// TIA Portal project "通信" (V16)

(* hardware
DEVICE "S7-1200 station_1"  S7-1200 Station
   slot 0: "Rack_0"  S7-1200 Rack  Rack  V1.0
   slot 1: "PLC_1"  CPU 1214C DC/DC/DC  6ES7 214-1AG40-0XB0  V4.4
*)

// ===== PLC "PLC_1"  CPU 1214C DC/DC/DC =====

VAR_GLOBAL   // PLC tag table "默认变量表"
   "System_Byte" AT %MB1 : Byte;
   "FirstScan" AT %M1.0 : Bool;
   "DiagStatusUpdate" AT %M1.1 : Bool;
   "AlwaysTRUE" AT %M1.2 : Bool;
   "AlwaysFALSE" AT %M1.3 : Bool;
   "Clock_Byte" AT %MB0 : Byte;
   "Clock_10Hz" AT %M0.0 : Bool;
   "Clock_5Hz" AT %M0.1 : Bool;
   "Clock_2.5Hz" AT %M0.2 : Bool;
   "Clock_2Hz" AT %M0.3 : Bool;
   "Clock_1.25Hz" AT %M0.4 : Bool;
   "Clock_1Hz" AT %M0.5 : Bool;
   "Clock_0.625Hz" AT %M0.6 : Bool;
   "Clock_0.5Hz" AT %M0.7 : Bool;
   "发完成" AT %M100.0 : Bool;
   "接完成" AT %M101.0 : Bool;
END_VAR

DATA_BLOCK "接受DB"   // DB1
{ S7_Optimized_Access := 'FALSE' }
VERSION : 0.1
   VAR
      其他 : Array[0..1] of Byte;
      接收 : Array[0..20] of Byte;
   END_VAR
BEGIN
END_DATA_BLOCK

DATA_BLOCK "传输DB"   // DB2
{ S7_Optimized_Access := 'FALSE' }
VERSION : 0.1
   VAR
      传送DB : Array[0..20] of Byte;
   END_VAR
BEGIN
END_DATA_BLOCK

DATA_BLOCK "数据块_1"   // DB5
{ S7_Optimized_Access := 'FALSE' }
VERSION : 0.1
   VAR
      "1" : Bool;
   END_VAR
BEGIN
END_DATA_BLOCK

ORGANIZATION_BLOCK "Main"   // OB1, LAD, ProgramCycle
TITLE = "Main Program Sweep (Cycle)"
{ S7_Optimized_Access := 'TRUE' }
VERSION : 0.1
   VAR_INPUT
      Initial_Call : Bool;   // Initial call of this OB
      Remanence : Bool;   // =True, if remanent data are available
   END_VAR
BEGIN

REGION Network 2: 传输
   // 先传输，之后接受，在
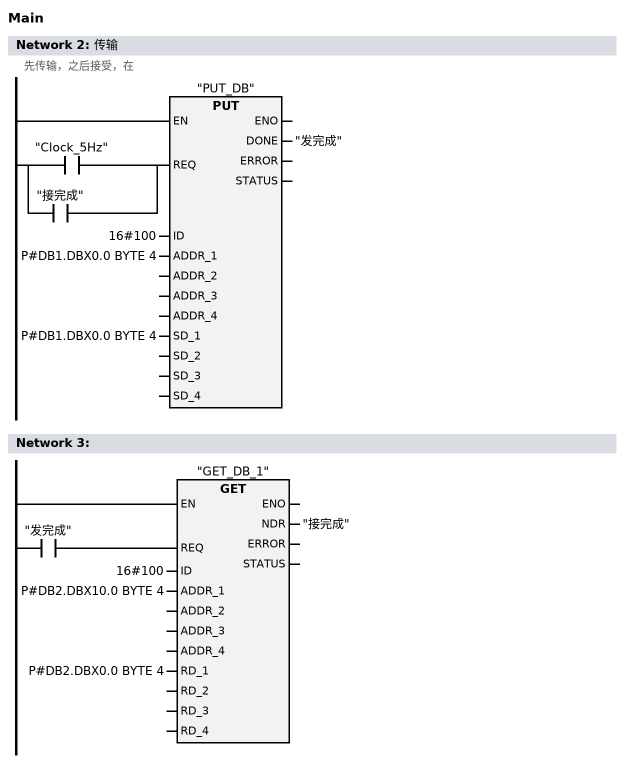
   "PUT_DB"(REQ := "Clock_5Hz" OR "接完成",   // PUT
            ID := 16#100,
            ADDR_1 := P#DB1.DBX0.0 BYTE 4,
            SD_1 := P#DB1.DBX0.0 BYTE 4,
            DONE => "发完成");
END_REGION

REGION Network 3
   "GET_DB_1"(REQ := "发完成",   // GET
              ID := 16#100,
              ADDR_1 := P#DB2.DBX10.0 BYTE 4,
              RD_1 := P#DB2.DBX0.0 BYTE 4,
              NDR => "接完成");
END_REGION
END_ORGANIZATION_BLOCK